Fanuc KAREL source: kd00029.KL

-- PROVISIONAL review KL for V770-1; original PC SHA256 808bf42232e35d2e58d6985c791cc406046fdc85138a2d2e9cc0b92201f7b7ff
-- Incomplete behavior may be omitted. Consult companion uncertainty JSON. Do not deploy.
PROGRAM KD00029
%NOLOCKGROUP
VAR
  I : INTEGER
  J : INTEGER
  B : BOOLEAN
  R : REAL
  S : STRING[80]
BEGIN
  -- UNRESOLVED_PC offsets 5-21; opcodes 9D,81,18,9C,12,22,9D,13,04
  -- UNRESOLVED_PC offsets 26-30; opcodes 7F
END KD00029
